PROGRAM OP90_SCN_ENB
VAR
END_VAR

OP90_HOMING();
OP90_MANUAL();
OP90_AUTO();

END_PROGRAM

(* stored: Version 1.1.0.1, ProductVersion 3.1.4024.11
   POU OP90_SCN_ENB: Id {7da84601-3039-4545-87fb-943c88b29f9c}, SpecialFunc None *)
